VAR_GLOBAL CONSTANT
	///ctrl commands definitions
	///specific commands >200 - every command has to be a even number
	cCMD_ADDALARM: INT := 202;
	cCMD_REMOVEALARM: INT := 204;
	///ctrl specific states definitions
	cSTA_ADDALARM: INT := AGS_CmdState.cCMD_ADDALARM;
	cSTA_REMOVEALARM: INT := AGS_CmdState.cCMD_REMOVEALARM;
END_VAR

(* stored: Version 1.1.0.1, ProductVersion 3.1.0.26
   GVL AGS_CmdState: Id {f20d22cb-2713-45e8-91f9-9230d2a5ef3c} *)
